// TIA Portal V19 export
DATA_BLOCK "TestInstLPythagorean"   // DB10002
// #@AutoGenerated
// stored: InstanceOfName LPythagorean, InstanceOfType FB
"LPythagorean"
   // VAR_INPUT
   //    "a" : Real;
   //    "b" : Real;
   // END_VAR
   // VAR_OUTPUT
   //    c : Real;
   //    valid : Bool;
   // END_VAR
BEGIN
END_DATA_BLOCK
